FUNCTION_BLOCK FB_Sum
VAR_INPUT
END_VAR
VAR_OUTPUT
END_VAR
VAR
END_VAR

{attribute 'TcRpcEnable'}
METHOD Sum : INT
VAR_INPUT
	A : INT;
	B : INT;
END_VAR
Sum := A+B;
END_METHOD

END_FUNCTION_BLOCK

(* stored: Version 1.1.0.1, ProductVersion 3.1.4024.12
   POU FB_Sum: Id {d4a8a67c-7d1e-46df-8367-1d72bd208e23}, SpecialFunc None
   Method Sum: Id {c024cfb3-3163-4978-a4cf-a92ae02489d2} *)
